PROGRAM WaterTankFilling
VAR
	fbTank			: FB_Tank;
	fbPump			: FB_Pump;
	fbDrainValve	: FB_DrainValve;
END_VAR

(*EXECUTE FBs*)
	fbPump.Execute();
	fbDrainValve.Execute();
	
(*PUMP - UPDATE LEVEL UNTIL LEVEL HIGH*)
	IF fbPump.bIsOn THEN
		IF NOT fbTank.bLevelHigh THEN
			fbTank.UpdateLevel(
				rFlowRate 			:= fbPump.rFlowRate, 
				rTimeStepSec		:= TO_REAL(TO_LREAL(_TaskInfo[GETCURTASKINDEXEX()].CycleTime) / 10_000_000));
		ELSIF fbTank.bLevelHigh THEN
			fbPump.Stop();
		END_IF
	END_IF

(*DRAIN VALVE - UPDATE LEVEL UNTIL TANK EMPTY*)
	IF fbDrainValve.bIsOn THEN
		IF NOT fbTank.bIsEmpty THEN
			fbTank.UpdateLevel(
					rFlowRate 		:= fbDrainValve.rFlowRate,
					rTimeStepSec	:= TO_REAL(TO_LREAL(_TaskInfo[GETCURTASKINDEXEX()].CycleTime) / 10_000_000));
		ELSE
			fbDrainValve.Stop();
		END_IF
	END_IF

END_PROGRAM

(* stored: Version 1.1.0.1, ProductVersion 3.1.4024.12
   POU WaterTankFilling: Id {6bc3bd89-2ad3-415d-8f59-322664583d9b}, SpecialFunc None *)
